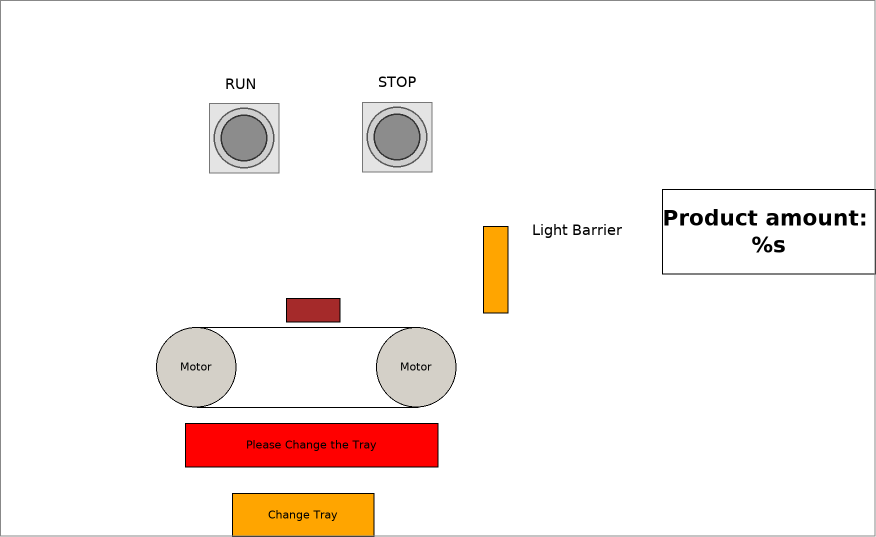
VISUALIZATION Visualization  // 876x537
    PushSwitchLed (209,103 70x70), variable: MAIN.StartPb, behaviour: TAP, style: Switch-PushSwitchLed-Gray
    PushSwitchLed (362,102 70x70), variable: MAIN.StopPB, behaviour: TAP, style: Switch-PushSwitchLed-Gray
    Rectangle (662,189 214x85), "Product amount: %s", text variable: MAIN.ProductCounter
    Ellipse (156,327 80x80), "Motor", colour toggle: MAIN.Motor
    Label (200,69 82x30), "RUN"
    Label (356,67 82x30), "STOP"
    Ellipse (376,327 80x80), "Motor", colour toggle: MAIN.Motor
    Line (197,407) (418,407)
    Line (197,327) (418,327)
    Rectangle (286,298 54x24)
    Rectangle (483,226 25x87), angle 48
        tap MAIN.LightBarrierSensor
    Label (519,215 116x30), "Light Barrier"
    Rectangle (232,493 142x44), "Change Tray", colour toggle: MAIN.ProductCnt.Q
        tap MAIN.TrayChange
    Rectangle (185,423 253x44), "Please Change the Tray", colour toggle: MAIN.ProductCnt.Q, invisible if: NOT MAIN.ProductCnt.Q
END_VISUALIZATION

(* stored: Version 1.1.0.1, ProductVersion 3.1.4024.15
   Visu Visualization: Id {69d51047-4eea-488d-8145-05668e8b9574} *)
